SUBAPPLICATION FullTwoStateCtrl (* Subapplication Type *)
  (* Standard: 61499-2 *)
  (* Version 1.0, 2020-07-27, AK120569 *)
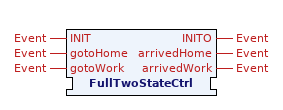
  EVENT_INPUT
    INIT;
    gotoHome;
    gotoWork;
  END_EVENT
  EVENT_OUTPUT
    INITO;
    arrivedHome;
    arrivedWork;
  END_EVENT
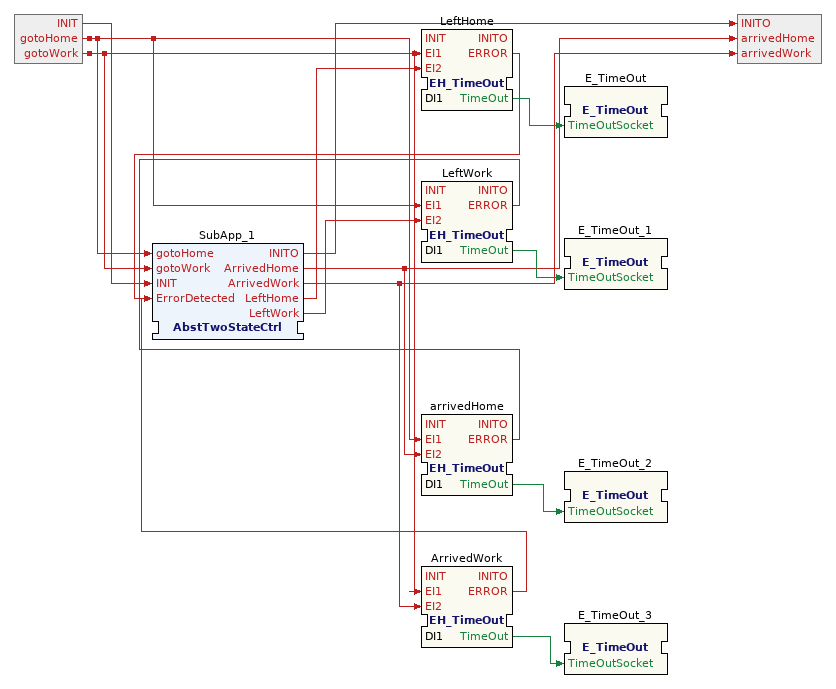
  FBS
    LeftHome : EH_TimeOut;
    LeftWork : EH_TimeOut;
    arrivedHome : EH_TimeOut;
    ArrivedWork : EH_TimeOut;
    E_TimeOut : E_TimeOut;
    E_TimeOut_1 : E_TimeOut;
    E_TimeOut_2 : E_TimeOut;
    E_TimeOut_3 : E_TimeOut;
  END_FBS
  SUBAPPS
    SubApp_1 : AbstTwoStateCtrl;
  END_SUBAPPS
  EVENT_CONNECTIONS
    gotoHome TO SubApp_1.gotoHome;
    gotoWork TO SubApp_1.gotoWork;
    INIT TO SubApp_1.INIT;
    SubApp_1.INITO TO INITO;
    SubApp_1.ArrivedHome TO arrivedHome;
    SubApp_1.ArrivedWork TO arrivedWork;
    SubApp_1.LeftHome TO LeftHome.EI2;
    gotoWork TO LeftHome.EI1;
    gotoHome TO LeftWork.EI1;
    SubApp_1.LeftWork TO LeftWork.EI2;
    gotoHome TO arrivedHome.EI1;
    SubApp_1.ArrivedHome TO arrivedHome.EI2;
    gotoWork TO ArrivedWork.EI1;
    SubApp_1.ArrivedWork TO ArrivedWork.EI2;
    ArrivedWork.ERROR TO SubApp_1.ErrorDetected;
    arrivedHome.ERROR TO SubApp_1.ErrorDetected;
    LeftWork.ERROR TO SubApp_1.ErrorDetected;
    LeftHome.ERROR TO SubApp_1.ErrorDetected;
  END_CONNECTIONS
  ADAPTER_CONNECTIONS
    LeftHome.TimeOut TO E_TimeOut.TimeOutSocket;
    LeftWork.TimeOut TO E_TimeOut_1.TimeOutSocket;
    arrivedHome.TimeOut TO E_TimeOut_2.TimeOutSocket;
    ArrivedWork.TimeOut TO E_TimeOut_3.TimeOutSocket;
  END_CONNECTIONS
END_SUBAPPLICATION
